FUNCTION_BLOCK E_SPLIT (* Template for an empty basic function block *)
  (* Standard: 61499-1 Annex A; Classification: event function block; Function: Split one event into two events; Description: Copyright (c) 2017 fortiss GmbH This program and the accompanying materials are made available under the terms of the Eclipse Public License 2.0 which is available at https://www.eclipse.org/legal/epl-2.0/ SPDX-License-Identifier: EPL-2.0 *)
  (* Version 1.0, 2017, Alois Zoitl, fortiss GmbH, initial API and implementation and/or initial documentation *)
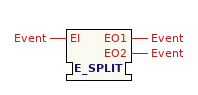
  EVENT_INPUT
    EI;
  END_EVENT
  EVENT_OUTPUT
    EO1;
    EO2;
  END_EVENT
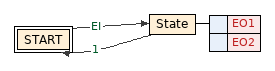
  EC_STATES
    START; (* Initial State *)
    State : -> EO1, -> EO2; (* "" *)
  END_STATES
  EC_TRANSITIONS
    START TO State := EI;
    State TO START := 1;
  END_TRANSITIONS
END_FUNCTION_BLOCK
